TYPE UDT_CylinderOutput :
STRUCT
	ValveIn: BOOL;
	ValveOut: BOOL;
	Error: BOOL;
	ErrorID: DINT;
END_STRUCT
END_TYPE

(* stored: Version 1.1.0.1, ProductVersion 3.1.4022.16
   DUT UDT_CylinderOutput: Id {273c19d9-c397-431c-9c57-cd8e26e9bbf1} *)
